PROGRAM ERROR
VAR
	StopX_a : MC_Stop;
	StopX_b : MC_Stop;
	StopY : MC_Stop;
	StopZ : MC_Stop;

END_VAR

// https://infosys.beckhoff.com/english.php?content=../content/1033/tccncmcplatform_fb/html/mcstop.htm&id=
// start stop pause continue

StopX_a(Axis := gvl.As_Xa,
		Execute := GVL.StopALL);

StopX_b(Axis := gvl.As_Xb,
		Execute := GVL.StopALL);

StopY(Axis := gvl.As_Y,
		Execute := GVL.StopALL);
		
StopZ(Axis := gvl.As_Z,
		Execute := GVL.StopALL);

END_PROGRAM

(* stored: Version 1.1.0.1, ProductVersion 3.1.4022.17
   POU ERROR: Id {8d68ba2e-431f-4b62-8370-2a49d23c7211}, SpecialFunc None *)
